FUNCTION_BLOCK E_SPLIT_4
  (* Standard: 61499-2 *)
  (* Version 11-09-13, slimrte *)
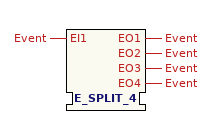
  EVENT_INPUT
    EI1;
  END_EVENT
  EVENT_OUTPUT
    EO1;
    EO2;
    EO3;
    EO4;
  END_EVENT
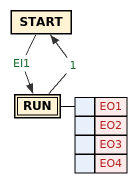
  EC_STATES
    RUN : -> EO1, -> EO2, -> EO3, -> EO4;
    START;
  END_STATES
  EC_TRANSITIONS
    START TO RUN := EI1;
    RUN TO START := 1;
  END_TRANSITIONS
END_FUNCTION_BLOCK
